// LS Electric XG5000 project: 커스텀통신시도2
// PLC LSPLC
// module base 0 slot 0: 입출력 모듈:XBC-DR32H (DC 24V 입력, 릴레이 출력 32점)

PROGRAM NewProgram (task: 스캔 프로그램)

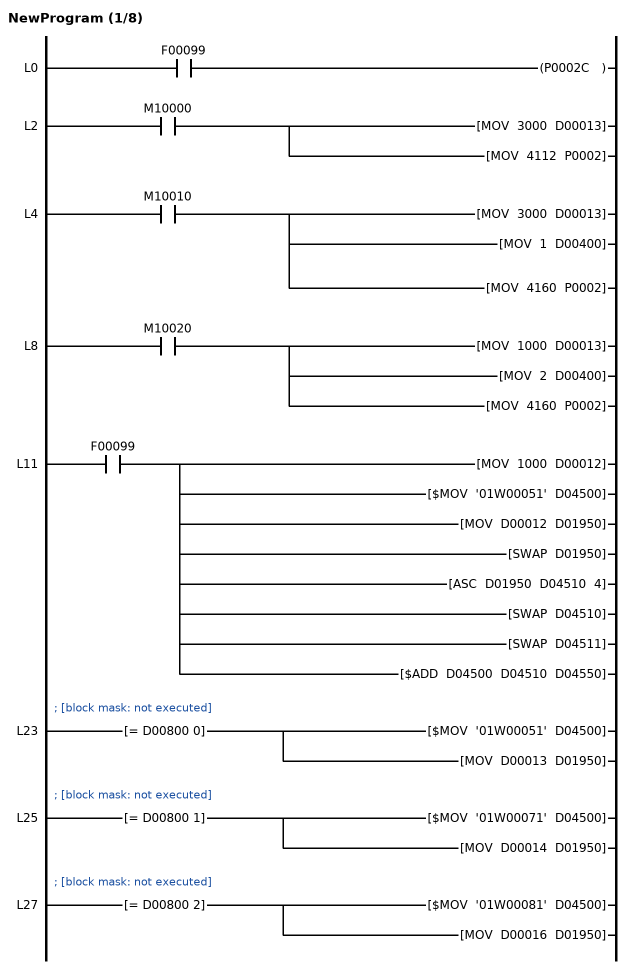
; L0
LOAD      F00099
OUT       P0002C
; L2
LOAD      M10000
MOV       3000 D00013
MOV       4112 P0002
; L4
LOAD      M10010
MOV       3000 D00013
MOV       1 D00400
MOV       4160 P0002
; L8
LOAD      M10020
MOV       1000 D00013
MOV       2 D00400
MOV       4160 P0002
; L11
LOAD      F00099
MOV       1000 D00012
$MOV      '01W00051' D04500
MOV       D00012 D01950
SWAP      D01950
ASC       D01950 D04510 4
SWAP      D04510
SWAP      D04511
$ADD      D04500 D04510 D04550
; L23 (block mask: not executed)
LOAD=     D00800 0
$MOV      '01W00051' D04500
MOV       D00013 D01950
; L25 (block mask: not executed)
LOAD=     D00800 1
$MOV      '01W00071' D04500
MOV       D00014 D01950
; L27 (block mask: not executed)
LOAD=     D00800 2
$MOV      '01W00081' D04500
MOV       D00016 D01950

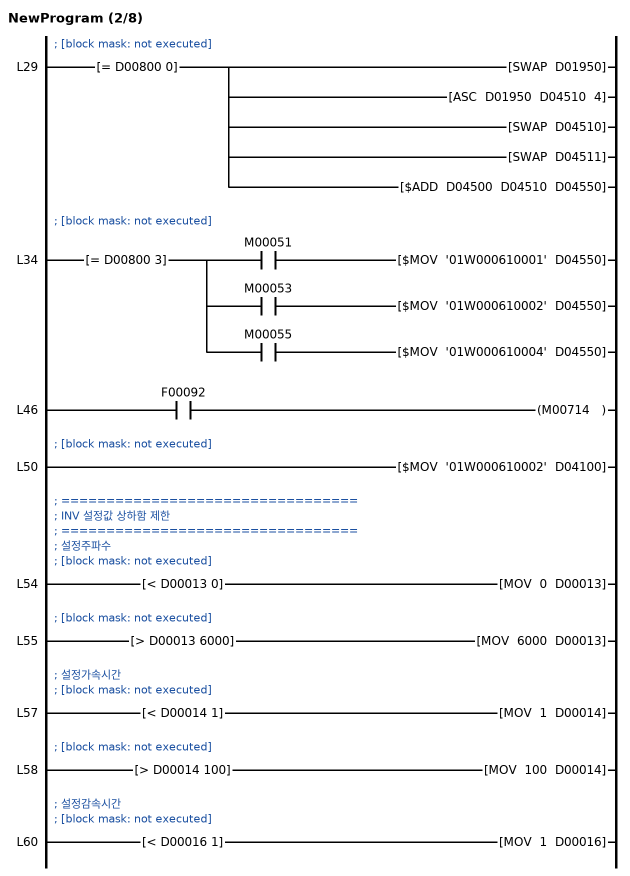
; L29 (block mask: not executed)
LOAD=     D00800 0
SWAP      D01950
ASC       D01950 D04510 4
SWAP      D04510
SWAP      D04511
$ADD      D04500 D04510 D04550
; L34 (block mask: not executed)
LOAD=     D00800 3
MPUSH
AND       M00051
$MOV      '01W000610001' D04550
MLOAD
AND       M00053
$MOV      '01W000610002' D04550
MPOP
AND       M00055
$MOV      '01W000610004' D04550
; L46
LOAD      F00092
OUT       M00714
; L50 (block mask: not executed)
$MOV      '01W000610002' D04100
// =================================
//    INV 설정값 상하함 제한
// =================================
// 설정주파수
; L54 (block mask: not executed)
LOAD<     D00013 0
MOV       0 D00013
; L55 (block mask: not executed)
LOAD>     D00013 6000
MOV       6000 D00013
// 설정가속시간
; L57 (block mask: not executed)
LOAD<     D00014 1
MOV       1 D00014
; L58 (block mask: not executed)
LOAD>     D00014 100
MOV       100 D00014
// 설정감속시간
; L60 (block mask: not executed)
LOAD<     D00016 1
MOV       1 D00016

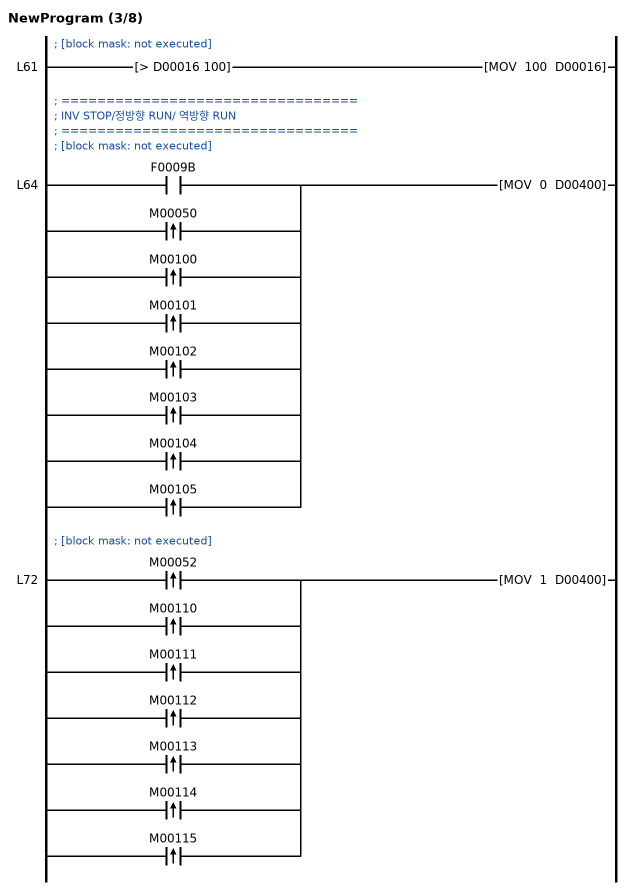
; L61 (block mask: not executed)
LOAD>     D00016 100
MOV       100 D00016
// =================================
//    INV STOP/정방향 RUN/ 역방향 RUN
// =================================
; L64 (block mask: not executed)
LOAD      F0009B
ORP       M00050
ORP       M00100
ORP       M00101
ORP       M00102
ORP       M00103
ORP       M00104
ORP       M00105
MOV       0 D00400
; L72 (block mask: not executed)
LOADP     M00052
ORP       M00110
ORP       M00111
ORP       M00112
ORP       M00113
ORP       M00114
ORP       M00115
MOV       1 D00400

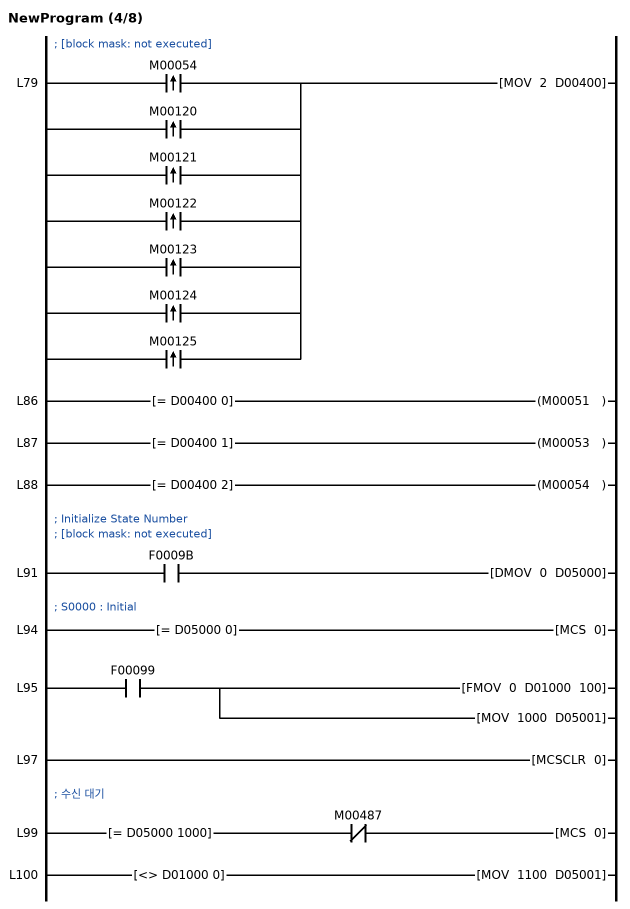
; L79 (block mask: not executed)
LOADP     M00054
ORP       M00120
ORP       M00121
ORP       M00122
ORP       M00123
ORP       M00124
ORP       M00125
MOV       2 D00400
; L86
LOAD=     D00400 0
OUT       M00051
; L87
LOAD=     D00400 1
OUT       M00053
; L88
LOAD=     D00400 2
OUT       M00054
// Initialize State Number
; L91 (block mask: not executed)
LOAD      F0009B
DMOV      0 D05000
// S0000 : Initial
; L94
LOAD=     D05000 0
MCS       0
; L95
LOAD      F00099
FMOV      0 D01000 100
MOV       1000 D05001
; L97
MCSCLR    0
// 수신 대기
; L99
LOAD=     D05000 1000
AND NOT   M00487
MCS       0
; L100
LOAD<>    D01000 0
MOV       1100 D05001

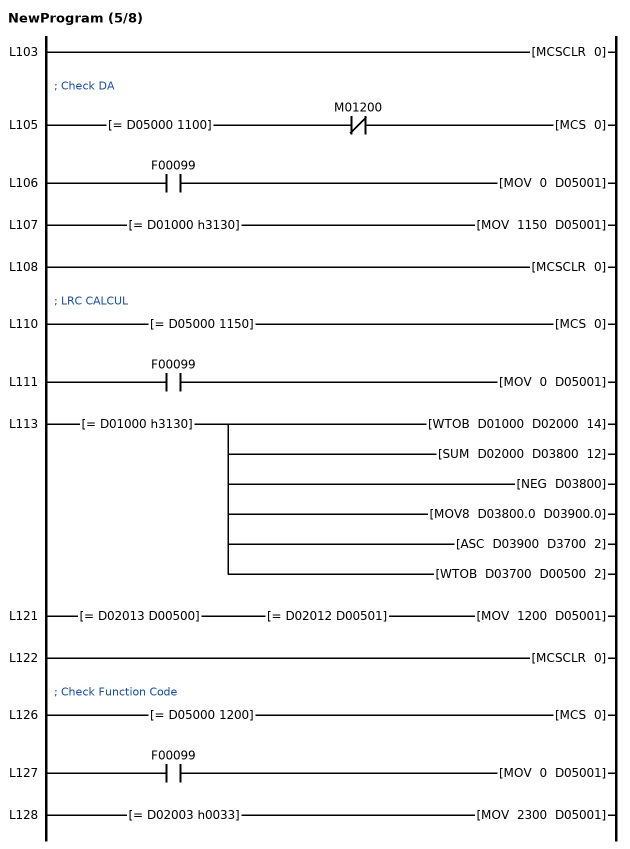
; L103
MCSCLR    0
// Check DA
; L105
LOAD=     D05000 1100
AND NOT   M01200
MCS       0
; L106
LOAD      F00099
MOV       0 D05001
; L107
LOAD=     D01000 h3130
MOV       1150 D05001
; L108
MCSCLR    0
// LRC CALCUL
; L110
LOAD=     D05000 1150
MCS       0
; L111
LOAD      F00099
MOV       0 D05001
; L113
LOAD=     D01000 h3130
WTOB      D01000 D02000 14
SUM       D02000 D03800 12
NEG       D03800
MOV8      D03800.0 D03900.0
ASC       D03900 D3700 2
WTOB      D03700 D00500 2
; L121
LOAD=     D02013 D00500
AND=      D02012 D00501
MOV       1200 D05001
; L122
MCSCLR    0
// Check Function Code
; L126
LOAD=     D05000 1200
MCS       0
; L127
LOAD      F00099
MOV       0 D05001
; L128
LOAD=     D02003 h0033
MOV       2300 D05001

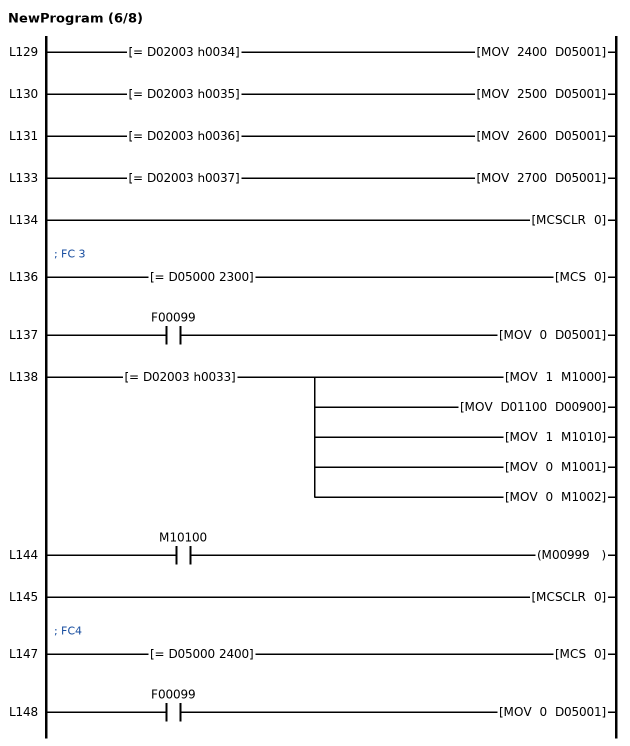
; L129
LOAD=     D02003 h0034
MOV       2400 D05001
; L130
LOAD=     D02003 h0035
MOV       2500 D05001
; L131
LOAD=     D02003 h0036
MOV       2600 D05001
; L133
LOAD=     D02003 h0037
MOV       2700 D05001
; L134
MCSCLR    0
// FC 3
; L136
LOAD=     D05000 2300
MCS       0
; L137
LOAD      F00099
MOV       0 D05001
; L138
LOAD=     D02003 h0033
MOV       1 M1000
MOV       D01100 D00900
MOV       1 M1010
MOV       0 M1001
MOV       0 M1002
; L144
LOAD      M10100
OUT       M00999
; L145
MCSCLR    0
// FC4
; L147
LOAD=     D05000 2400
MCS       0
; L148
LOAD      F00099
MOV       0 D05001

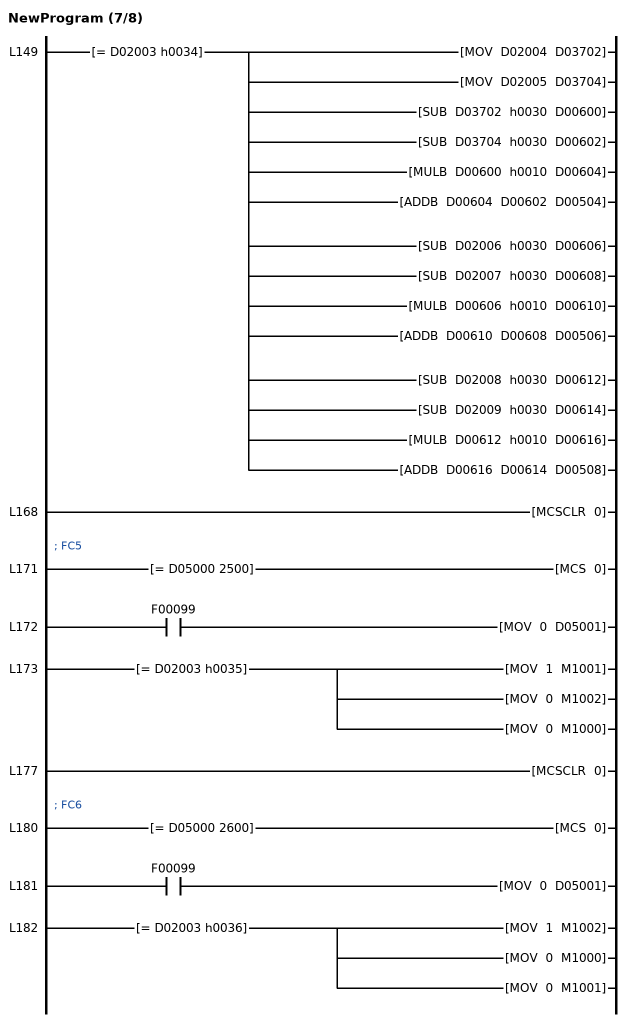
; L149
LOAD=     D02003 h0034
MOV       D02004 D03702
MOV       D02005 D03704
SUB       D03702 h0030 D00600
SUB       D03704 h0030 D00602
MULB      D00600 h0010 D00604
ADDB      D00604 D00602 D00504
SUB       D02006 h0030 D00606
SUB       D02007 h0030 D00608
MULB      D00606 h0010 D00610
ADDB      D00610 D00608 D00506
SUB       D02008 h0030 D00612
SUB       D02009 h0030 D00614
MULB      D00612 h0010 D00616
ADDB      D00616 D00614 D00508
; L168
MCSCLR    0
// FC5
; L171
LOAD=     D05000 2500
MCS       0
; L172
LOAD      F00099
MOV       0 D05001
; L173
LOAD=     D02003 h0035
MOV       1 M1001
MOV       0 M1002
MOV       0 M1000
; L177
MCSCLR    0
// FC6
; L180
LOAD=     D05000 2600
MCS       0
; L181
LOAD      F00099
MOV       0 D05001
; L182
LOAD=     D02003 h0036
MOV       1 M1002
MOV       0 M1000
MOV       0 M1001

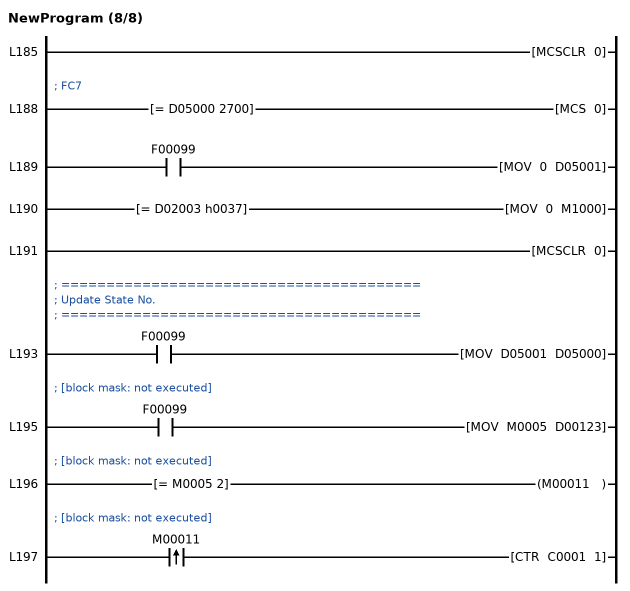
; L185
MCSCLR    0
// FC7
; L188
LOAD=     D05000 2700
MCS       0
; L189
LOAD      F00099
MOV       0 D05001
; L190
LOAD=     D02003 h0037
MOV       0 M1000
; L191
MCSCLR    0
// ========================================
// Update State No.
// ========================================
; L193
LOAD      F00099
MOV       D05001 D05000
; L195 (block mask: not executed)
LOAD      F00099
MOV       M0005 D00123
; L196 (block mask: not executed)
LOAD=     M0005 2
OUT       M00011
; L197 (block mask: not executed)
LOADP     M00011
CTR       C0001 1